// TIA Portal V17 export
// export: Created 2025-03-07T09:19:06.6503875Z, ExportSetting WithDefaults, DisplayName Totally Integrated Automation Portal, DisplayVersion V17 Update 8, DisplayName TIA Portal Openness, DisplayVersion V17 Update 8, DisplayName TIA Portal Version Control Interface, DisplayVersion V17, DisplayName SINAMICS Startdrive Advanced, DisplayVersion V17 SP2, DisplayName SINAMICS Startdrive G110M, G120, G120C, G120D, G120P, G115D, DisplayVersion V17 SP2, DisplayName SINAMICS Startdrive G130, G150, S120, S150, SINAMICS MV, S210, DisplayVersion V17 SP2, DisplayName STEP 7 Professional, DisplayVersion V17 Update 8, DisplayName SINUMERIK ONE STEP 7 Toolbox, DisplayVersion V17 Update 12, DisplayName SINUMERIK 840D sl STEP 7 Toolbox, DisplayVersion V17 Update 12, DisplayName STEP 7 Safety, DisplayVersion V17 Update 6, DisplayName WinCC Advanced, DisplayVersion V17 Update 8
DATA_BLOCK "DB16010_MEASURE_SENSORS_CALIBRATION_STATUS"   // DB16010
{ S7_Optimized_Access := 'FALSE'; DB_Accessible_From_OPC_UA := 'FALSE' }
VERSION : 0.1
// stored: AutoNumber false, DBAccessibleFromOPCUA false, DBAccessibleFromWebserver true, IsOnlyStoredInLoadMemory false, IsWriteProtectedInAS false
   VAR RETAIN
      HMI : Struct
         U01_FORCE_CALIBRATION : Bool;   // UNIT 01 PERFILOMETER FORCE CALIBRATION
         U01_CANCEL_FORCE_CALIBRATION : Bool;   // UNIT 01 PERFILOMETER CANCEL FORCE CALIBRATION
         U01_STA_3_CALIBRATION_CYCLE_REQ : Bool;   // UNIT 01 PERFILOMETER STATION 3 CALIBRATION CYCLE REQUEST
         U01_STA_0_TURN_REQ : Bool;   // UNIT 01 STATION 0 CYCLE REQUEST
         U01_START_CAM_CALIBRATION : Bool;   // UNIT 01 COAXIAL CAMERA START CALIBRATION BUTTON
         U01_START_CAM_ALIGNMENT : Bool;   // UNIT 01 COAXIAL CAMERA START ALIGNMENT BUTTON
         U01_STOP_CAM_METHODS : Bool;   // UNIT 01 COAXIAL CAMERA STOP METHODS BUTTON
         U01_CAM_SAVE_RECORDING : Bool;   // UNIT 01 COAXIAL CAMERA SAVE RECORDINGS BUTON
         U01_FIXTURE_SELECTED : Byte := 16#1;   // UNIT 01 FIXTURE SELECTED
         U02_FORCE_CALIBRATION : Bool;   // UNIT 02 PERFILOMETER FORCE CALIBRATION
         U02_CANCEL_FORCE_CALIBRATION : Bool;   // UNIT 02 PERFILOMETER CANCEL FORCE CALIBRATION
         U02_STA_2_CALIBRATION_CYCLE_REQ : Bool;   // UNIT 02 PERFILOMETER STATION 2 CALIBRATION CYCLE REQUEST
         U02_STA_3_CALIBRATION_CYCLE_REQ : Bool;   // UNIT 02 PERFILOMETER STATION 3 CALIBRATION CYCLE REQUEST
         U02_STA_0_TURN_REQ : Bool;   // UNIT 02 STATION 0 CYCLE REQUEST
         U02_START_CAM_CALIBRATION : Bool;   // UNIT 02 COAXIAL CAMERA START CALIBRATION BUTTON
         U02_START_CAM_ALIGNMENT : Bool;   // UNIT 02 COAXIAL CAMERA START ALIGNMENT BUTTON
         U02_STOP_CAM_METHODS : Bool;   // UNIT 02 COAXIAL CAMERA STOP METHODS BUTTON
         U02_CAM_SAVE_RECORDING : Bool;   // UNIT 02 COAXIAL CAMERA SAVE RECORDINGS BUTON
         U02_FIXTURE_SELECTED : Byte := 16#1;   // UNIT 02 FIXTURE SELECTED
         U03_FORCE_CALIBRATION : Bool;   // UNIT 02 PERFILOMETER FORCE CALIBRATION
         U03_CANCEL_FORCE_CALIBRATION : Bool;   // UNIT 02 PERFILOMETER CANCEL FORCE CALIBRATION
         U03_FACE_SELECTED : Byte := 16#1;   // UNIT 01 FIXTURE SELECTED
      END_STRUCT;
      U01_STA3_MEAS : Struct
         FIXTURE_1_STATUS : Int;   // FIXTURE 1 SENSOR UNIT 01 STATION 3 CALIBRATION MISSING
         FIXTURE_2_STATUS : Int;   // FIXTURE 2 SENSOR UNIT 01 STATION 3 CALIBRATION MISSING
         FIXTURE_3_STATUS : Int;   // FIXTURE 3 SENSOR UNIT 01 STATION 3 CALIBRATION MISSING
         FIXTURE_4_STATUS : Int;   // FIXTURE 4 SENSOR UNIT 01 STATION 3 CALIBRATION MISSING
      END_STRUCT;
      U02_STA2_MEAS : Struct
         FIXTURE_1_STATUS : Int;   // FIXTURE 1 SENSOR UNIT 02 STATION 2 CALIBRATION MISSING
         FIXTURE_2_STATUS : Int;   // FIXTURE 2 SENSOR UNIT 02 STATION 2 CALIBRATION MISSING
         FIXTURE_3_STATUS : Int;   // FIXTURE 3 SENSOR UNIT 02 STATION 2 CALIBRATION MISSING
         FIXTURE_4_STATUS : Int;   // FIXTURE 4 SENSOR UNIT 02 STATION 2 CALIBRATION MISSING
      END_STRUCT;
      U02_STA3_MEAS : Struct
         FIXTURE_1_STATUS : Int;   // FIXTURE 1 SENSOR UNIT 02 STATION 3 CALIBRATION MISSING
         FIXTURE_2_STATUS : Int;   // FIXTURE 2 SENSOR UNIT 02 STATION 3 CALIBRATION MISSING
         FIXTURE_3_STATUS : Int;   // FIXTURE 3 SENSOR UNIT 02 STATION 3 CALIBRATION MISSING
         FIXTURE_4_STATUS : Int;   // FIXTURE 4 SENSOR UNIT 02 STATION 3 CALIBRATION MISSING
      END_STRUCT;
      U03_STA_MEAS_MEAS_R : Struct
         FIXTURE_1_STATUS : Int;   // FIXTURE 1 SENSOR UNIT 03 STATION MEAS FACE R CALIBRATION MISSING
      END_STRUCT;
      U03_STA_MEAS_MEAS_N : Struct
         FIXTURE_1_STATUS : Int;   // FIXTURE 1 SENSOR UNIT 03 STATION MEAS FACE N CALIBRATION MISSING
      END_STRUCT;
      UNIT_01_AUX { ExternalAccessible := 'False'; ExternalVisible := 'False'; ExternalWritable := 'False'} : Struct
         FIXTURE_1_FORCE_CALIB_MEM { ExternalAccessible := 'False'; ExternalVisible := 'False'; ExternalWritable := 'False'} : Bool;   // FIXTURE 1 SENSOR UNIT 01 STATION 3 FORCE CALIBRATION MEMORY
         FIXTURE_2_FORCE_CALIB_MEM { ExternalAccessible := 'False'; ExternalVisible := 'False'; ExternalWritable := 'False'} : Bool;   // FIXTURE 2 SENSOR UNIT 01 STATION 3 FORCE CALIBRATION MEMORY
         FIXTURE_3_FORCE_CALIB_MEM { ExternalAccessible := 'False'; ExternalVisible := 'False'; ExternalWritable := 'False'} : Bool;   // FIXTURE 3 SENSOR UNIT 01 STATION 3 FORCE CALIBRATION MEMORY
         FIXTURE_4_FORCE_CALIB_MEM { ExternalAccessible := 'False'; ExternalVisible := 'False'; ExternalWritable := 'False'} : Bool;   // FIXTURE 4 SENSOR UNIT 01 STATION 3 FORCE CALIBRATION MEMORY
      END_STRUCT;
      UNIT_02_AUX : Struct
         STATION_2 : Struct
            FIXTURE_1_FORCE_CALIB_MEM : Bool;   // FIXTURE 1 SENSOR UNIT 02 STATION 2 FORCE CALIBRATION MEMORY
            FIXTURE_2_FORCE_CALIB_MEM : Bool;   // FIXTURE 2 SENSOR UNIT 02 STATION 2 FORCE CALIBRATION MEMORY
            FIXTURE_3_FORCE_CALIB_MEM : Bool;   // FIXTURE 3 SENSOR UNIT 02 STATION 2 FORCE CALIBRATION MEMORY
            FIXTURE_4_FORCE_CALIB_MEM : Bool;   // FIXTURE 4 SENSOR UNIT 02 STATION 2 FORCE CALIBRATION MEMORY
         END_STRUCT;
         STATION_3 : Struct
            FIXTURE_1_FORCE_CALIB_MEM : Bool;   // FIXTURE 1 SENSOR UNIT 02 STATION 3 FORCE CALIBRATION MEMORY
            FIXTURE_2_FORCE_CALIB_MEM : Bool;   // FIXTURE 2 SENSOR UNIT 02 STATION 3 FORCE CALIBRATION MEMORY
            FIXTURE_3_FORCE_CALIB_MEM : Bool;   // FIXTURE 3 SENSOR UNIT 02 STATION 3 FORCE CALIBRATION MEMORY
            FIXTURE_4_FORCE_CALIB_MEM : Bool;   // FIXTURE 4 SENSOR UNIT 02 STATION 3 FORCE CALIBRATION MEMORY
         END_STRUCT;
         UNIT_01_AUX { ExternalAccessible := 'False'; ExternalVisible := 'False'; ExternalWritable := 'False'} : Struct
            FIXTURE_1_FORCE_CALIB_MEM { ExternalAccessible := 'False'; ExternalVisible := 'False'; ExternalWritable := 'False'} : Bool;   // FIXTURE 1 SENSOR UNIT 01 STATION 3 FORCE CALIBRATION MEMORY
            FIXTURE_2_FORCE_CALIB_MEM { ExternalAccessible := 'False'; ExternalVisible := 'False'; ExternalWritable := 'False'} : Bool;   // FIXTURE 2 SENSOR UNIT 01 STATION 3 FORCE CALIBRATION MEMORY
            FIXTURE_3_FORCE_CALIB_MEM { ExternalAccessible := 'False'; ExternalVisible := 'False'; ExternalWritable := 'False'} : Bool;   // FIXTURE 3 SENSOR UNIT 01 STATION 3 FORCE CALIBRATION MEMORY
            FIXTURE_4_FORCE_CALIB_MEM { ExternalAccessible := 'False'; ExternalVisible := 'False'; ExternalWritable := 'False'} : Bool;   // FIXTURE 4 SENSOR UNIT 01 STATION 3 FORCE CALIBRATION MEMORY
         END_STRUCT;
      END_STRUCT;
      UNIT_03_AUX { ExternalAccessible := 'False'; ExternalVisible := 'False'; ExternalWritable := 'False'} : Struct
         FACE_A_FORCE_CALIB_MEM { ExternalAccessible := 'False'; ExternalVisible := 'False'; ExternalWritable := 'False'} : Bool;   // FACE A SENSOR UNIT 03 FORCE CALIBRATION MEMORY
         FACE_B_FORCE_CALIB_MEM { ExternalAccessible := 'False'; ExternalVisible := 'False'; ExternalWritable := 'False'} : Bool;   // FACE B SENSOR UNIT 03 FORCE CALIBRATION MEMORY
      END_STRUCT;
   END_VAR
BEGIN
END_DATA_BLOCK
